// Notice: Each state has a corresponding controller, which has a fixed index.
// Add the new state at the end and update the total num
TYPE E_MasterArmState :
(
	MasterArmState_Error := 1,
	MasterArmState_Init :=2,
	MasterArmState_Home :=3,
	MasterArmState_Standby :=4,
	MasterArmState_Matching :=5,
	MasterArmState_Ready :=6,
	MasterArmState_MasterSlave :=7,
	MasterArmState_Clutch :=8,
	MasterArmState_Endoscope :=9,
	MasterArmState_Cart := 10,
	MasterArmState_GravityCali := 11,
	MasterArmState_Test :=12,
	MasterArmState_Disable :=13,
	MasterArmState_Performance :=14,
	MasterArmState_Selfcheck := 15,
	MasterArmState_PowerOff := 16,
	MasterArmState_GravityBiasCali := 17,
	
	MasterArmState_PrecisionTest :=50,
	MasterArmState_TestCycle :=51,
	MasterArmState_TestFriction:=52,
	MasterArmState_TestResponse:=53,
	MasterArmState_TestDragFree:=54,
	MasterArmState_ManiTest :=55,
	MasterArmState_armCali :=56,
	
	MasterArmState_totalNum :=MasterArmState_armCali
);
END_TYPE

(* stored: Version 1.1.0.1, ProductVersion 3.1.4024.11
   DUT E_MasterArmState: Id {1772d389-f98f-4390-a8fe-c1a65ee5f75e} *)
